FUNCTION_BLOCK T_RoboConnect_SetToolDigitalOutput_ReturnsTrueOutput EXTENDS T_UnitTestBase
VAR
  robot : I_RoboConnect;
  timeOutTimer : TON;
  targetDO : UINT;
  myTestState, prevState :
    (INIT,
    ARRANGE,
    ACT,
    ASSERT) := INIT;
  expected, actual : BOOL;
  counter : UINT;
  returnedTask : I_Task;
  resultTask : I_BoolResultTask;
END_VAR

CASE myTestState OF
  INIT:
    StateChanged();
    myTestState := ARRANGE;

  ARRANGE:
    IF StateChanged() THEN
      expected := TRUE;
      robot.Connect();
    END_IF

    IF robot.Connected THEN
      myTestState := ACT;
    END_IF

  ACT:
    robot.SetToolDigitalOutput(targetDO, TRUE, task => returnedTask);
    myTestState := ASSERT;

  ASSERT:

    IF timeOutTimer.Q THEN
      actual := robot.GetToolDigitalOutput(targetDO, task => resultTask);
      assertion.AssertEquals_BOOL(expected, actual, 'actual := robot.GetToolDigitalOutput(targetDO, task => resultTask)');
      TestFinished();
      myTestState := INIT;

    END_IF

END_CASE

timeOutTimer(IN := myTestState = ASSERT);

METHOD FB_init : BOOL
VAR_INPUT
  bInitRetains : BOOL; // if TRUE, the retain variables are initialized (warm start / cold start)
  bInCopyCode : BOOL; // if TRUE, the instance afterwards gets moved into the copy code (online change)
  TestSuite : tcl_SimpleUnitTestLibrary.I_TestSuite;
  robot : I_TcRobot;
  timeout : TIME;
  targetDo : UINT;
END_VAR
THIS^.robot := robot;
THIS^.timeOutTimer.PT := timeout;
THIS^.targetDo := targetDo;
END_METHOD

METHOD PRIVATE StateChanged : BOOL
IF  myTestState = prevState THEN
  RETURN;
END_IF

prevState := myTestState;
StateChanged := TRUE;
END_METHOD

METHOD WaitForCycles : BOOL
VAR_INPUT
  maxCount : UINT;
END_VAR
counter := counter + 1;

IF counter = maxCount THEN
  counter := 0;
  WaitForCycles := TRUE;
END_IF
END_METHOD

END_FUNCTION_BLOCK

(* stored: Version 1.1.0.1
   POU T_TcRobot_SetToolDigitalOutput_ReturnsTrueOutput: Id {f1401383-e3b9-4426-85fd-872a75782e33}, SpecialFunc None
   Method FB_init: Id {2c6f643c-0e4d-4e26-9653-51401b119ca0}
   Method StateChanged: Id {9dfc1334-eab7-4422-920e-e45206bd298a}
   Method WaitForCycles: Id {00522937-c4ee-4b21-8129-422ae3c0d30f} *)
